% RSLogix 500 project LIFT- PLC.RSS, saved by version 8.30.00.16 %
PROJECT "UNTITLED"    % processor: MicroLogix 1000 %

PROGRAM FILES
  LAD 2 "MAIN_PROG"  5 rungs
  LAD 3 "USER_FAULT"  1 rungs
  LAD 4 "HSC_INT"  1 rungs
  LAD 5 "STI_INT"  1 rungs
  LAD 6, 7, 8, 9, 10, 11, 12, 13, 14, 15, 16: only END

DATA FILES
  O0 OUTPUT  1 elements
  I1 INPUT  2 elements
  S2 STATUS  33 elements
  B3 BINARY  32 elements
  T4 TIMER  40 elements
  C5 COUNTER  32 elements
  R6 CONTROL  16 elements
  N7 INTEGER  105 elements

LADDER 2 "MAIN_PROG"
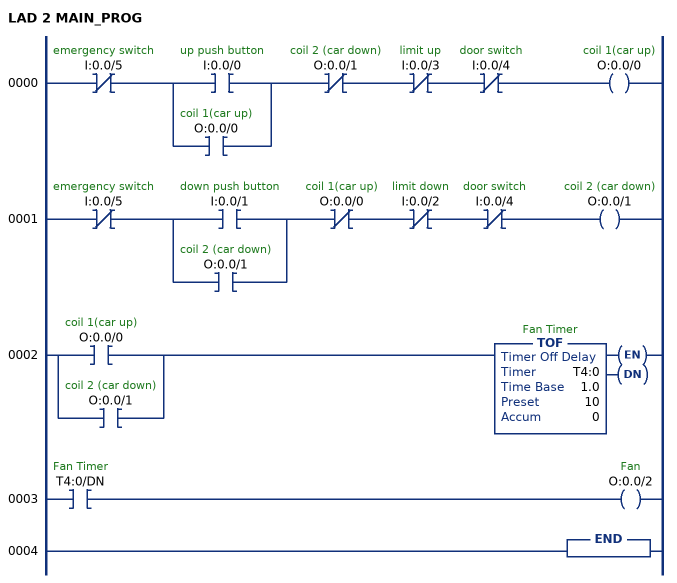
% Rung: 0 %
SOR XIO I:0.0/5 BST XIC I:0.0/0 NXB XIC O:0.0/0 BND XIO O:0.0/1 XIO I:0.0/3 XIO I:0.0/4 OTE O:0.0/0 EOR
%   I:0.0/5  "emergency switch" %
%   I:0.0/0  "up push button" %
%   O:0.0/0  "coil 1(car up)" %
%   O:0.0/1  "coil 2 (car down)" %
%   I:0.0/3  "limit up" %
%   I:0.0/4  "door switch" %
% Rung: 1 %
SOR XIO I:0.0/5 BST XIC I:0.0/1 NXB XIC O:0.0/1 BND XIO O:0.0/0 XIO I:0.0/2 XIO I:0.0/4 OTE O:0.0/1 EOR
%   I:0.0/5  "emergency switch" %
%   I:0.0/1  "down push button" %
%   O:0.0/1  "coil 2 (car down)" %
%   O:0.0/0  "coil 1(car up)" %
%   I:0.0/2  "limit down" %
%   I:0.0/4  "door switch" %
% Rung: 2 %
SOR BST XIC O:0.0/0 NXB XIC O:0.0/1 BND TOF T4:0 1.0 10 0 EOR
%   O:0.0/0  "coil 1(car up)" %
%   O:0.0/1  "coil 2 (car down)" %
%   T4:0  "Fan Timer" %
% Rung: 3 %
SOR XIC T4:0/DN OTE O:0.0/2 EOR
%   T4:0  "Fan Timer" %
%   O:0.0/2  "Fan" %
% Rung: 4 %
SOR END EOR

OTHER DOCUMENTED ADDRESSES
  I:0.0/6  "emergency switch"
  O:0.0/3  "a1"
  T4:0/0  "Timer"

DATA TABLE (non-zero values as saved)
DATA T4
% .PRE .ACC %
% T4:0 % 10 0
